FUNCTION_BLOCK WP_OR (* Basic Function Block Type *)
  (* Standard: 61499-2 *)
  (* Version 0.0, 2/7/2012, XPMUser, nxtControl GmbH, Template *)
  PACKAGE Main;
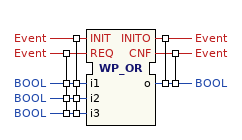
  EVENT_INPUT
    INIT WITH i1, i3, i2; (* Initialization Request *)
    REQ WITH i1, i2, i3; (* Normal Execution Request *)
  END_EVENT
  EVENT_OUTPUT
    INITO WITH o; (* Initialization Confirm *)
    CNF WITH o; (* Execution Confirmation *)
  END_EVENT
  VAR_INPUT
    i1 : BOOL; (* Input event qualifier *)
    i2 : BOOL;
    i3 : BOOL;
  END_VAR
  VAR_OUTPUT
    o : BOOL; (* Output event qualifier *)
  END_VAR
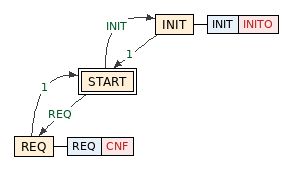
  EC_STATES
    START; (* Initial State *)
    INIT : INIT -> INITO; (* Initialization *)
    REQ : REQ -> CNF; (* Normal execution *)
  END_STATES
  EC_TRANSITIONS
    START TO INIT := INIT;
    INIT TO START := 1;
    START TO REQ := REQ;
    REQ TO START := 1;
  END_TRANSITIONS
  ALGORITHM INIT IN ST: (* Initialization algorithm *)
IF i1 = TRUE OR i2 = TRUE OR i3 = TRUE THEN
    o := TRUE;
ELSE
    o := FALSE;
END_IF;
  END_ALGORITHM
  ALGORITHM REQ IN ST: (* Normally executed algorithm *)
IF i1 = TRUE OR i2 = TRUE OR i3 = TRUE THEN
    o := TRUE;
ELSE
    o := FALSE;
END_IF;
  END_ALGORITHM
END_FUNCTION_BLOCK
